// TIA Portal V21 export
// export: Created 2026-09-27T08:23:38.8834043Z, ExportSetting None
ORGANIZATION_BLOCK "Spike_Startup"   // OB100, SCL, Startup
TITLE = "Complete Restart"
{ S7_Optimized_Access := 'TRUE' }
// stored: SetENOAutomatically false
   VAR_INPUT
      LostRetentive : Bool;   // True if retentive data are lost
      LostRTC : Bool;   // True if date and time are lost
   END_VAR
BEGIN
END_ORGANIZATION_BLOCK
